ABB RobotStudio station: robotmanipulator.rsstn

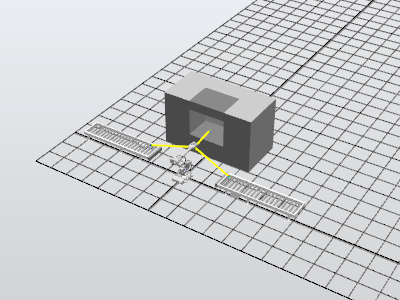
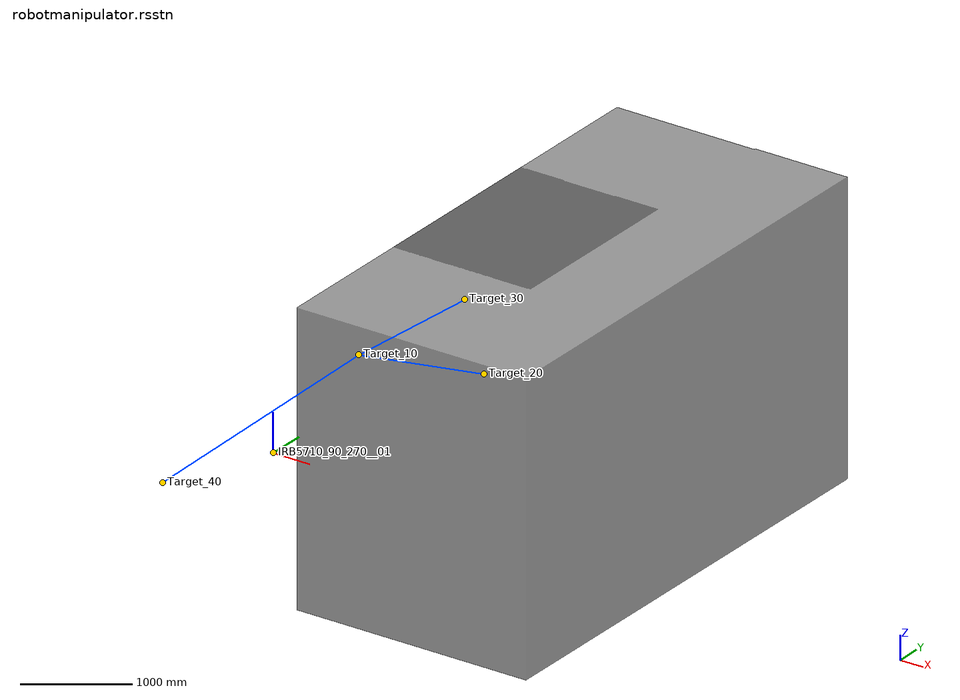
[picture v1: parts stored in the station drawn from their meshes, with robot base, taught points and paths (robot models come from the ABB library and are not in the file)]
Station Bitirme (saved by RobotStudio 25.1.11167.1)
Controller Controller1
  mechanical unit ROB_1: IRB5710_90_270__01, 6 joints, base frame (0, 0, 0) mm
Layout (positions relative to the parent item):
  - IRB5710_90_270__01 [mechanism, from %ABB.RobotStudio.Models.IRB5710%\IRB5710_90_270__01.rslib] at (0, 0, 0) mm; joint values [0, -1.0024, 0.9804, 0, 1.5928, 3.1416] (rad or m)
  - Part_10 [part] at (-211.26, -50.93, 0) mm, size 1500 x 1500 x 3000 mm
  - Part_11 [part] at (-210.17, 3433.9, 0) mm, size 1500 x 1500 x 3000 mm
  - Part_12 [part], size 1500 x 2000 x 1000 mm
  - Part_14 [part] at (0, 0, -500) mm, size 1500 x 2000 x 500 mm
  - Part_15 [part], size 1000 x 5000 x 3000 mm
  - 950_4000_h2 [part, from %ABB.RobotStudio.Models.Conveyors%\Conveyor 950 4000 h2.rslib] at (892.32, 2114.91, 0) mm, rotated rx 0 ry 0 rz 90 deg
  - 950_4000 [part, from %ABB.RobotStudio.Models.Conveyors%\Conveyor 950 4000 h2.rslib] at (-26.71, -1959.27, 0) mm, rotated rx 0 ry 0 rz -90 deg
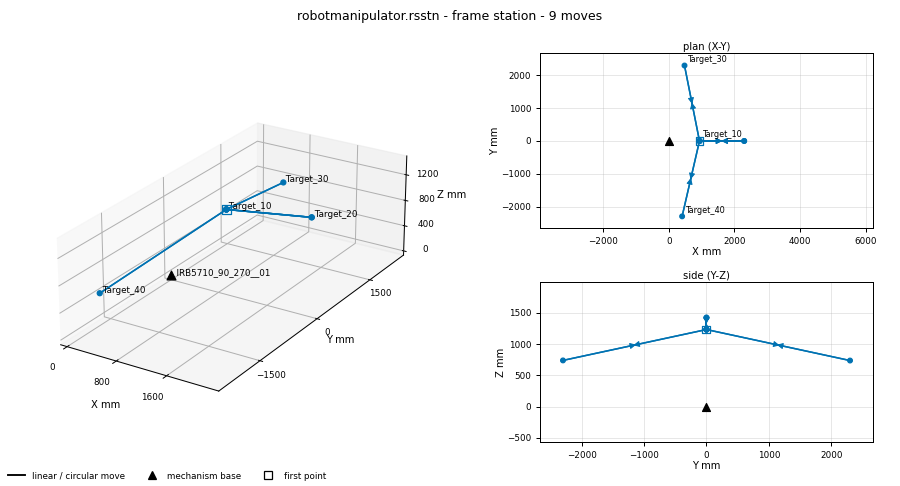
[picture p0: tool path of robotmanipulator.rsstn in frame station, 9 of 9 moves have a stored position in this frame; points joined in program order, loops and branches not executed]
Targets, tools, work objects and paths stored in the station, written as RAPID:
! task T_ROB1
MODULE Module1
  CONST robtarget Target_10:=[[935.072,0,1233.399],[0,1,0,0],[0,0,0,0],[9E+09,9E+09,9E+09,9E+09,9E+09,9E+09]];
  CONST robtarget Target_20:=[[2298.127,0,1424.481],[0,1,0,0],[0,0,2,0],[9E+09,9E+09,9E+09,9E+09,9E+09,9E+09]];
  CONST robtarget Target_30:=[[478.314,2300.29,736.735],[0,1,0,0],[0,0,2,0],[9E+09,9E+09,9E+09,9E+09,9E+09,9E+09]];
  CONST robtarget Target_40:=[[405.732,-2298.729,738.731],[0,1,0,0],[-1,0,1,0],[9E+09,9E+09,9E+09,9E+09,9E+09,9E+09]];
  CONST robtarget Target_10_1:=[[935.072,0,1233.399],[0,1,0,0],[0,0,0,0],[9E+09,9E+09,9E+09,9E+09,9E+09,9E+09]];
  CONST robtarget Target_10_2:=[[935.072,0,1233.399],[0,1,0,0],[0,0,0,0],[9E+09,9E+09,9E+09,9E+09,9E+09,9E+09]];
  CONST robtarget Target_10_3:=[[935.072,0,1233.399],[0,1,0,0],[0,0,0,0],[9E+09,9E+09,9E+09,9E+09,9E+09,9E+09]];
  PROC Path_10()
    MoveL Target_10,v1000,z100,tool0\WObj:=wobj0;
    MoveL Target_30,v1000,z100,tool0\WObj:=wobj0;
    WaitTime 0.7;
    MoveL Target_10_1,v1000,z100,tool0\WObj:=wobj0;
    MoveL Target_20,v1000,z100,tool0\WObj:=wobj0;
    WaitTime 0.7;
    MoveL Target_10_2,v1000,z100,tool0\WObj:=wobj0;
    WaitTime 2;
    MoveL Target_20,v1000,z100,tool0\WObj:=wobj0;
    WaitTime 0.7;
    MoveL Target_10_2,v1000,z100,tool0\WObj:=wobj0;
    MoveL Target_40,v1000,z100,tool0\WObj:=wobj0;
    WaitTime 0.7;
    MoveL Target_10_3,v1000,z100,tool0\WObj:=wobj0;
  ENDPROC
  PROC main()
    Path_10;
  ENDPROC
ENDMODULE

